// Mitsubishi GX Works2 project: PLCgroup16_updateeee   PLC: FX3G

// global labels: Global1
VAR_GLOBAL
  LampY7 AT Y007 : BOOL;
  SwitchX007 AT X007 : BOOL;
  M_EmptyInventory AT M0 : BOOL;
  X11_EmergencySwitch AT X011 : BOOL;
  SwitchY007 AT Y007 : BOOL;
  Sampling AT X001 : BOOL;
  Analog_Input AT D8280 : INT;
  check AT Y003 : BOOL;
END_VAR
VAR_GLOBAL CONSTANT
  Normalization : INT := 400;
END_VAR
VAR_GLOBAL
  Beer_Kind AT M1 : BOOL;
  Choose_beer_kind AT D1100 : REAL;
  choosing AT X006 : BOOL;
END_VAR
VAR_GLOBAL CONSTANT
  Limitt : REAL := 5.0;
END_VAR
VAR_GLOBAL
  test AT M1 : BOOL;
  Is_Pilsner AT M1 : BOOL;
  Yeast_Inventory AT D1102 : REAL;
END_VAR
VAR_GLOBAL CONSTANT
  Is_Enough_Yeast1 : REAL := 120.0;
END_VAR
VAR_GLOBAL
  Malt_Inventory AT D1104 : REAL;
END_VAR
VAR_GLOBAL CONSTANT
  Is_Enough_Malt : REAL := 6.0;
END_VAR
VAR_GLOBAL
  Hops_Inventory AT D1106 : REAL;
END_VAR
VAR_GLOBAL CONSTANT
  Is_Enough_Hops : REAL := 53.0;
END_VAR
VAR_GLOBAL
  Enough_Yeast AT M2 : BOOL;
  Enough_Malt AT M3 : BOOL;
  Enough_Hops AT M4 : BOOL;
  checking AT X003 : BOOL;
END_VAR
VAR_GLOBAL CONSTANT
  Is_Enough_Yeast2 : REAL := 150.0;
  Is_Enough_Malt2 : REAL := 12.0;
  Enough_Hops2 : REAL := 60.0;
END_VAR
VAR_GLOBAL
  Timer_Destenation AT TS1 : BOOL;
  Cooking_Light AT Y001 : BOOL;
  Timer_Coocking_Time_Finish AT TS1 : BOOL;
END_VAR
VAR_GLOBAL CONSTANT
  Cooking_Timer : REAL := 40.00;
END_VAR
VAR_GLOBAL
  Timer1 AT TC1 : BOOL;
END_VAR
VAR_GLOBAL CONSTANT
  Timer_Destenationn : INT := 40;
END_VAR
VAR_GLOBAL
  Start_Tsisa AT X005 : BOOL;
  Helping_Light AT M5 : BOOL;
  Timer_Blinking_Light_p AT TC2 : BOOL;
END_VAR
VAR_GLOBAL CONSTANT
  Blinking_Destenation1 : INT := 20;
END_VAR
VAR_GLOBAL
  Blinking_Destenationn AT TS2 : BOOL;
  First_Blinking_Light AT Y003 : BOOL;
  Timer_Blinking_Light_p2 AT TC3 : BOOL;
  Blinking_Destenationn2 AT TS3 : BOOL;
  Second_Blinking_Light AT Y004 : BOOL;
  Timer_Blinking_Light_l AT TC4 : BOOL;
END_VAR
VAR_GLOBAL CONSTANT
  Blinking_Destination3 : INT := 15;
END_VAR
VAR_GLOBAL
  Blinking_Destination_XD AT TS4 : BOOL;
  Timer_Blinking_Light_l2 AT TC5 : BOOL;
  Blinking_Destination_XDDDDD AT TS5 : BOOL;
  Storage_Phase AT X002 : BOOL;
END_VAR
VAR_GLOBAL CONSTANT
  Sub_Yeast : REAL := 120.0;
  Sub_Malt : REAL := 6.0;
  Sub_Hops : REAL := 53.0;
  Sub_Yeast1 : REAL := 150.0;
  Sub_Malt1 : REAL := 12.0;
  Sub_Hops1 : REAL := 60.0;
END_VAR
VAR_GLOBAL
  Pack_N_Save AT X000 : BOOL;
  Six_Six_Six AT Y002 : BOOL;
  Bottle_Counter AT CC0 : BOOL;
END_VAR
VAR_GLOBAL CONSTANT
  Full : INT := 6;
END_VAR
VAR_GLOBAL
  Bottle_Counter_Finish AT CS0 : BOOL;
  Fnish_Packing_Light AT Y002 : BOOL;
  SUBTRACT AT X004 : BOOL;
  Number_Of_Six_Packs AT D1108 : REAL;
END_VAR
VAR_GLOBAL CONSTANT
  Add_Created_Six_Pack : REAL := 1.0;
  Divide_To_Get_Decimal : REAL := 10.0;
END_VAR
VAR_GLOBAL
  Decimall_Six_Pack AT D1110 : REAL;
  Analog_Output AT D8282 : INT;
  Inventory_Watcher AT M5 : BOOL;
END_VAR
VAR_GLOBAL CONSTANT
  Normalization2 : INT := 40;
  Normalization22 : INT := 40;
  Multiplier : REAL := 40.0;
  Normalization_1 : INT := 400;
  kefel : REAL := 40.0;
  Zero : REAL;
  Zero_Word : INT;
END_VAR

// task Task_01 (event TRUE, interval 0, priority 31): POU_01

PROGRAM POU_01
VAR
  Sample : BOOL;
  Yeast_Float : REAL;
  Yeast : INT;
  Lowest_limit1 : BOOL;
END_VAR
VAR CONSTANT
  Is_Enough_Yeast : INT := 120;
END_VAR
VAR
  Cooking : BOOL;
END_VAR
(* structured ladder/FBD written out as ST: instructions are called as NAME(EN, inputs, outputs); _pN, _eN, _tN stand for wires *)
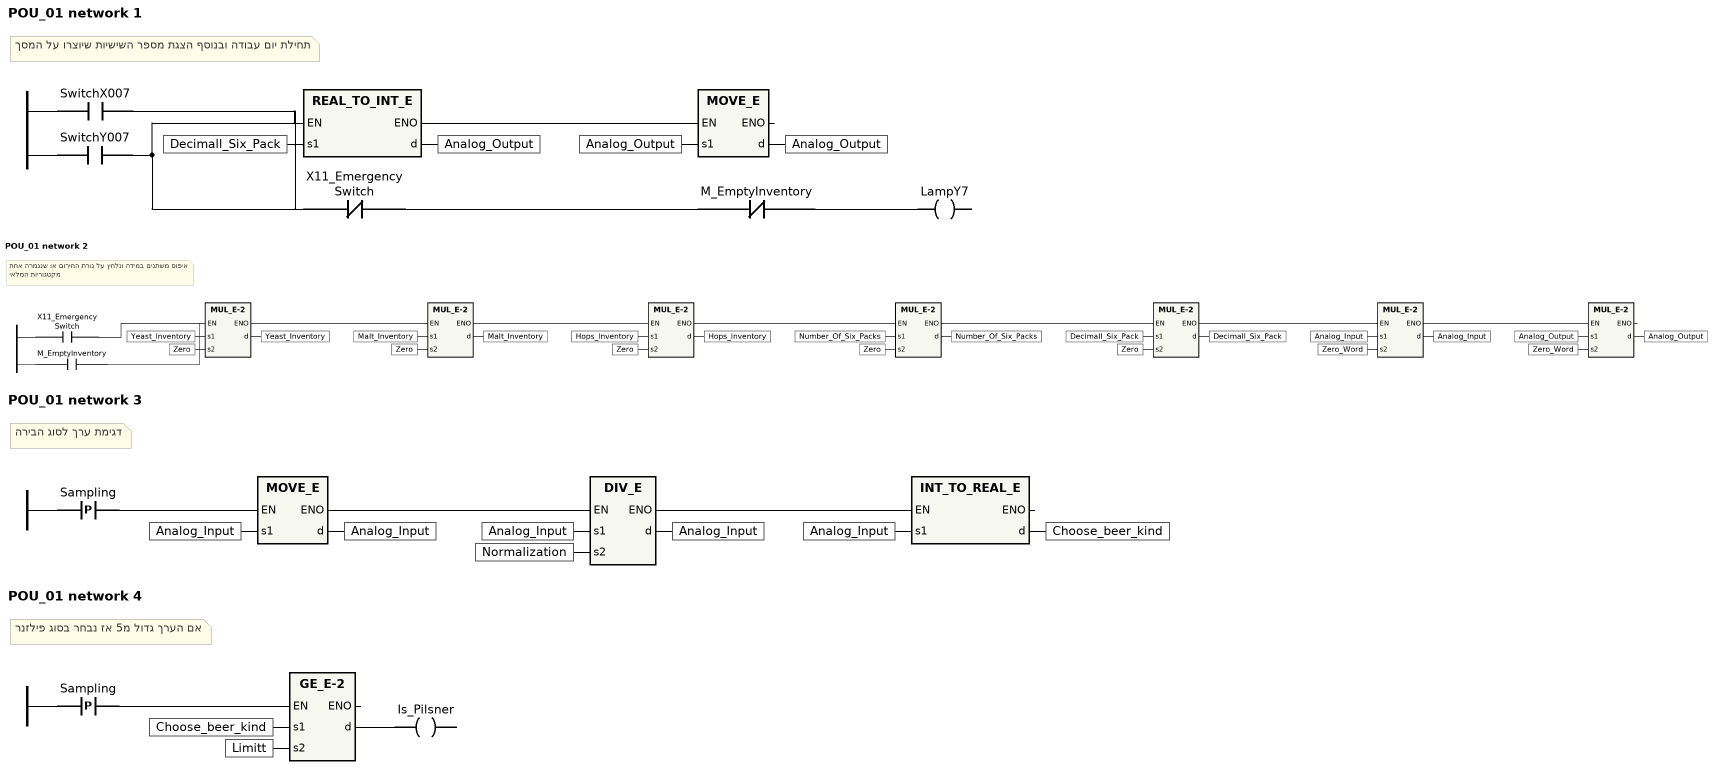
(* network 1 *)
(* תחילת יום עבודה ובנוסף הצגת מספר השישיות שיוצרו על המסך *)
_p1 := SwitchX007 OR SwitchY007;
LampY7 := _p1 AND NOT X11_EmergencySwitch AND NOT M_EmptyInventory;
_e2 := REAL_TO_INT_E(_p1, Decimall_Six_Pack, Analog_Output);
MOVE_E(_e2, Analog_Output, Analog_Output);
(* network 2 *)
(* איפוס משתנים במידה ונלחץ על נורת החירום או שנגמרה אחת מקטגוריות המלאי *)
_e1 := MUL_E(X11_EmergencySwitch OR M_EmptyInventory, Yeast_Inventory, Zero, Yeast_Inventory);
_e2 := MUL_E(_e1, Malt_Inventory, Zero, Malt_Inventory);
_e3 := MUL_E(_e2, Hops_Inventory, Zero, Hops_Inventory);
_e4 := MUL_E(_e3, Number_Of_Six_Packs, Zero, Number_Of_Six_Packs);
_e5 := MUL_E(_e4, Decimall_Six_Pack, Zero, Decimall_Six_Pack);
_e6 := MUL_E(_e5, Analog_Input, Zero_Word, Analog_Input);
MUL_E(_e6, Analog_Output, Zero_Word, Analog_Output);
(* network 3 *)
(* דגימת ערך לסוג הבירה *)
_e1 := MOVE_E(LDP(TRUE, Sampling), Analog_Input, Analog_Input);
_e2 := DIV_E(_e1, Analog_Input, Normalization, Analog_Input);
INT_TO_REAL_E(_e2, Analog_Input, Choose_beer_kind);
(* network 4 *)
(* אם הערך גדול מ5 אז נבחר בסוג פילזנר *)
GE_E(LDP(TRUE, Sampling), Choose_beer_kind, Limitt, _t1);
Is_Pilsner := _t1;
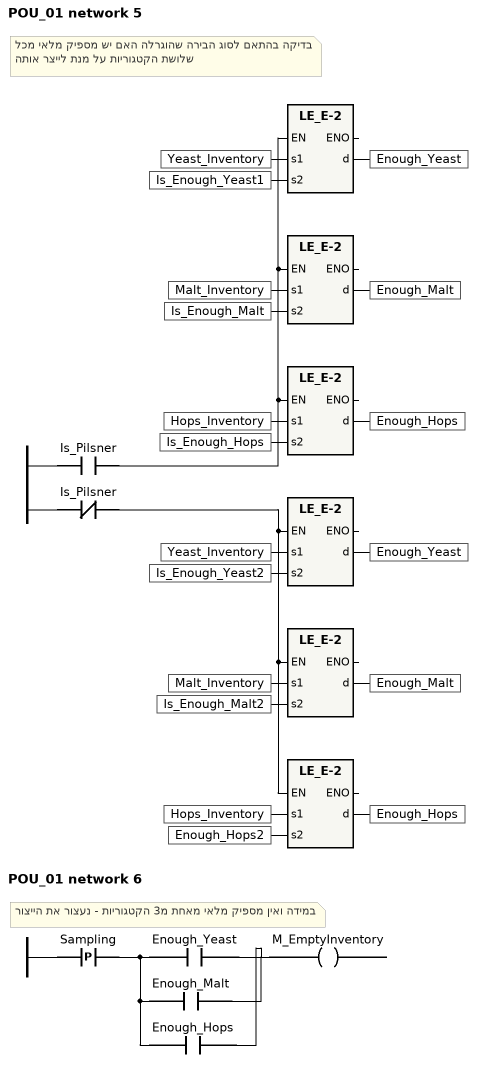
(* network 5 *)
(* בדיקה בהתאם לסוג הבירה שהוגרלה האם יש מספיק מלאי מכל שלושת הקטגוריות על מנת לייצר אותה *)
LE_E(Is_Pilsner, Yeast_Inventory, Is_Enough_Yeast1, Enough_Yeast);
LE_E(Is_Pilsner, Malt_Inventory, Is_Enough_Malt, Enough_Malt);
LE_E(Is_Pilsner, Hops_Inventory, Is_Enough_Hops, Enough_Hops);
_p1 := NOT Is_Pilsner;
LE_E(_p1, Yeast_Inventory, Is_Enough_Yeast2, Enough_Yeast);
LE_E(_p1, Malt_Inventory, Is_Enough_Malt2, Enough_Malt);
LE_E(_p1, Hops_Inventory, Enough_Hops2, Enough_Hops);
(* network 6 *)
(* במידה ואין מספיק מלאי מאחת מ3 הקטגוריות - נעצור את הייצור *)
_p1 := LDP(TRUE, Sampling);
M_EmptyInventory := (_p1 AND Enough_Yeast) OR (_p1 AND Enough_Malt) OR (_p1 AND Enough_Hops);
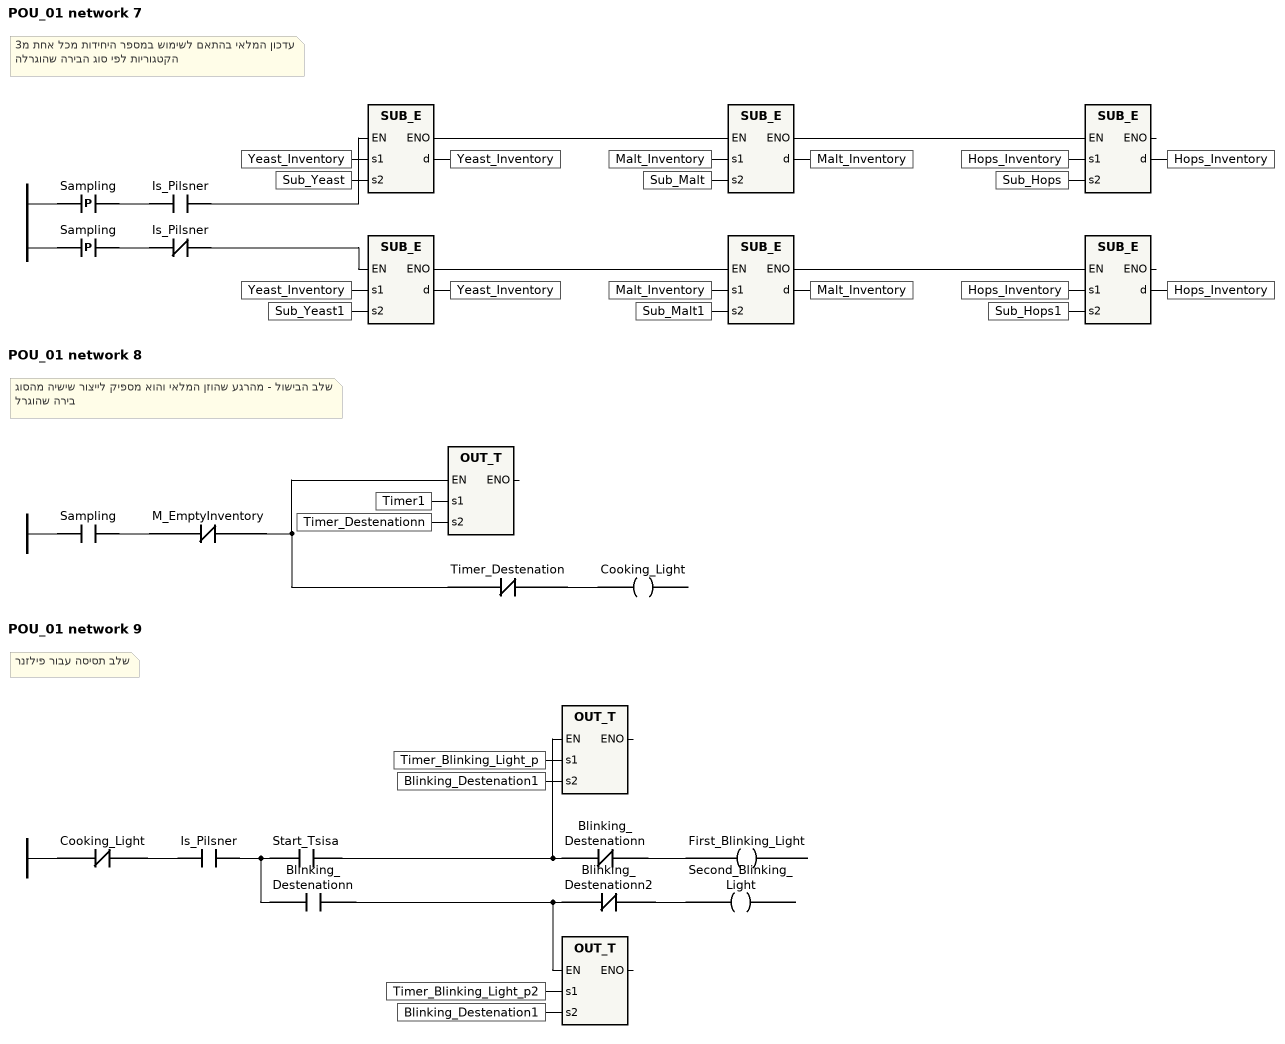
(* network 7 *)
(* עדכון המלאי בהתאם לשימוש במספר היחידות מכל אחת מ3 הקטגוריות לפי סוג הבירה שהוגרלה *)
_e1 := SUB_E(LDP(TRUE, Sampling) AND Is_Pilsner, Yeast_Inventory, Sub_Yeast, Yeast_Inventory);
_e2 := SUB_E(_e1, Malt_Inventory, Sub_Malt, Malt_Inventory);
SUB_E(_e2, Hops_Inventory, Sub_Hops, Hops_Inventory);
_e3 := SUB_E(LDP(TRUE, Sampling) AND NOT Is_Pilsner, Yeast_Inventory, Sub_Yeast1, Yeast_Inventory);
_e4 := SUB_E(_e3, Malt_Inventory, Sub_Malt1, Malt_Inventory);
SUB_E(_e4, Hops_Inventory, Sub_Hops1, Hops_Inventory);
(* network 8 *)
(* שלב הבישול - מהרגע שהוזן המלאי והוא מספיק לייצור שישיה מהסוג בירה שהוגרל *)
_p1 := Sampling AND NOT M_EmptyInventory;
OUT_T(_p1, Timer1, Timer_Destenationn);
Cooking_Light := _p1 AND NOT Timer_Destenation;
(* network 9 *)
(* שלב תסיסה עבור פילזנר *)
_p1 := NOT Cooking_Light AND Is_Pilsner;
_p2 := _p1 AND Start_Tsisa;
OUT_T(_p2, Timer_Blinking_Light_p, Blinking_Destenation1);
First_Blinking_Light := _p2 AND NOT Blinking_Destenationn;
_p3 := _p1 AND Blinking_Destenationn;
OUT_T(_p3, Timer_Blinking_Light_p2, Blinking_Destenation1);
Second_Blinking_Light := _p3 AND NOT Blinking_Destenationn2;
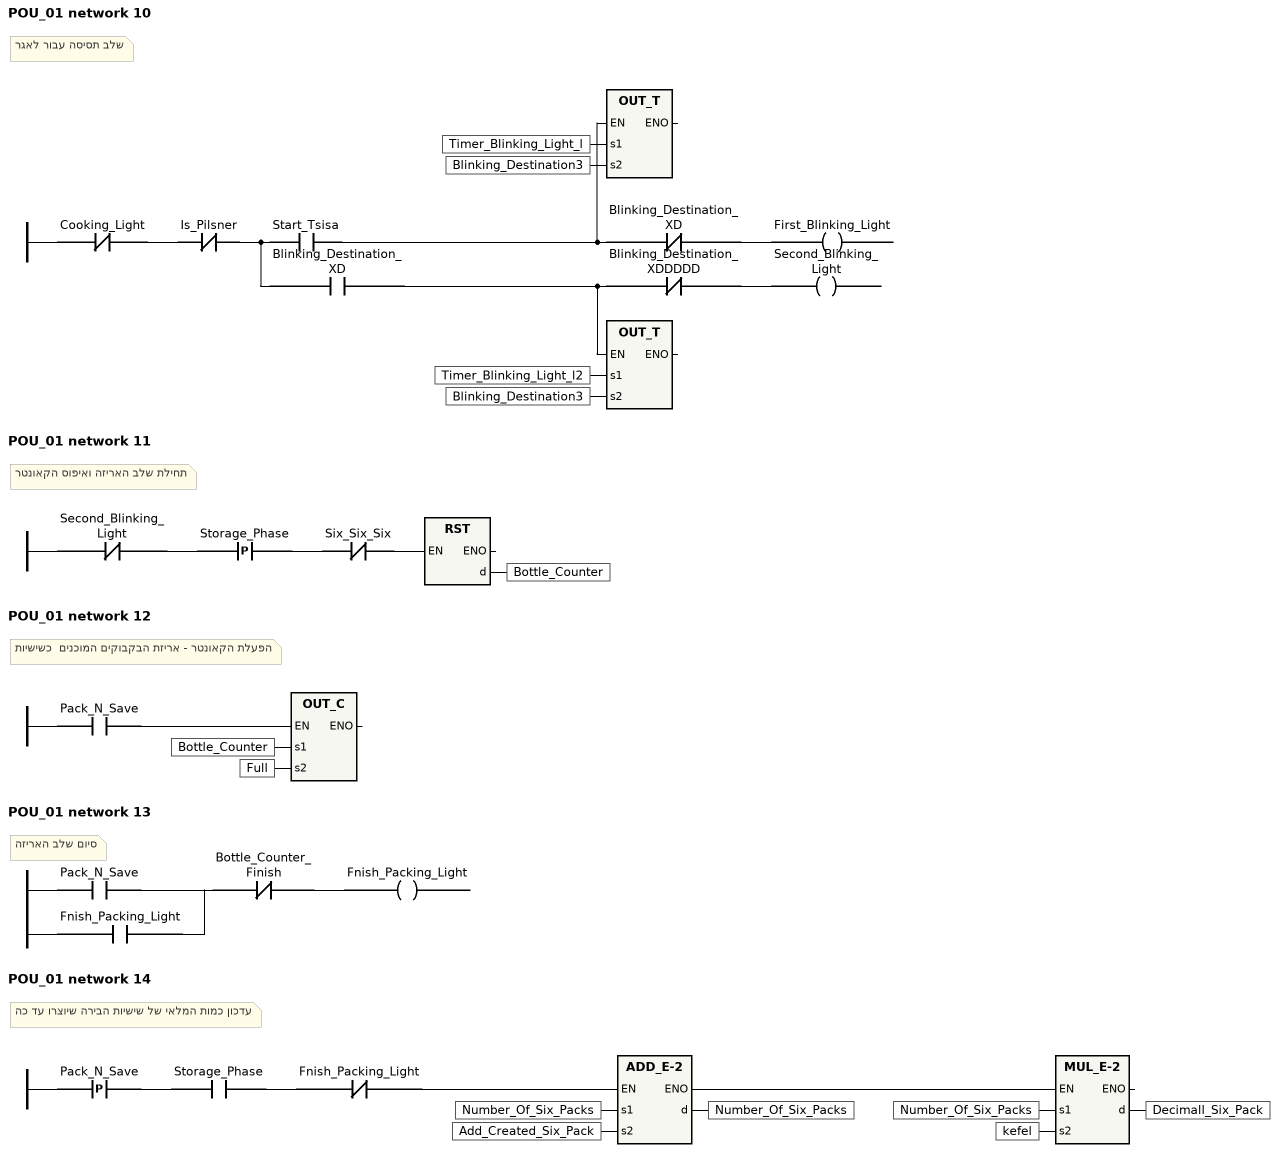
(* network 10 *)
(* שלב תסיסה עבור לאגר *)
_p1 := NOT Cooking_Light AND NOT Is_Pilsner;
_p2 := _p1 AND Start_Tsisa;
OUT_T(_p2, Timer_Blinking_Light_l, Blinking_Destination3);
First_Blinking_Light := _p2 AND NOT Blinking_Destination_XD;
_p3 := _p1 AND Blinking_Destination_XD;
OUT_T(_p3, Timer_Blinking_Light_l2, Blinking_Destination3);
Second_Blinking_Light := _p3 AND NOT Blinking_Destination_XDDDDD;
(* network 11 *)
(* תחילת שלב האריזה ואיפוס הקאונטר *)
RST(NOT Second_Blinking_Light AND LDP(TRUE, Storage_Phase) AND NOT Six_Six_Six, Bottle_Counter);
(* network 12 *)
(* הפעלת הקאונטר - אריזת הבקבוקים המוכנים  כשישיות *)
OUT_C(Pack_N_Save, Bottle_Counter, Full);
(* network 13 *)
(* סיום שלב האריזה *)
Fnish_Packing_Light := (Pack_N_Save OR Fnish_Packing_Light) AND NOT Bottle_Counter_Finish;
(* network 14 *)
(* עדכון כמות המלאי של שישיות הבירה שיוצרו עד כה *)
_e1 := ADD_E(LDP(TRUE, Pack_N_Save) AND Storage_Phase AND NOT Fnish_Packing_Light, Number_Of_Six_Packs, Add_Created_Six_Pack, Number_Of_Six_Packs);
MUL_E(_e1, Number_Of_Six_Packs, kefel, Decimall_Six_Pack);
END_PROGRAM
